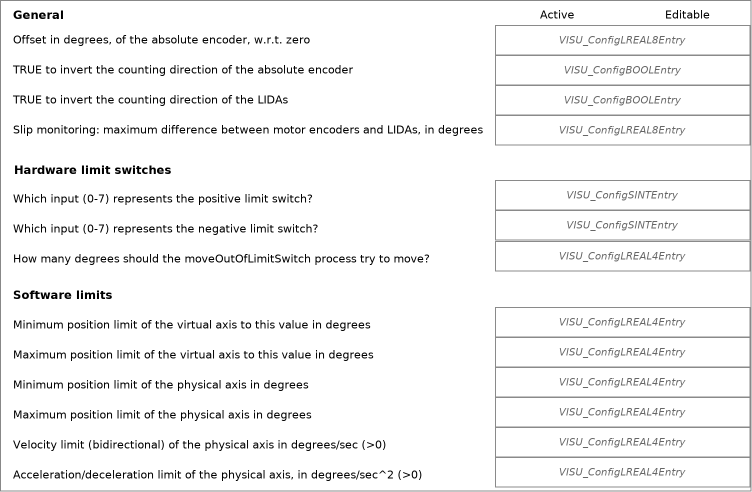
VISUALIZATION VISU_AxesConfig_Elevation_1  // 752x492
VAR_IN_OUT
    active : AxesElevationConfig;
    editable : AxesElevationConfig;
END_VAR
    Label (495,5 125x20), "Active"
    Label (625,5 125x20), "Editable"
    Label (10,25 360x30), "Offset in degrees, of the absolute encoder, w.r.t. zero"
    Frame (495,25 255x30)
        shows VISU_ConfigLREAL8Entry(active := active.absoluteEncoderOffset, editable := editable.absoluteEncoderOffset)
    Label (10,184 475x30), "Which input (0-7) represents the positive limit switch?"
    Label (10,214 475x30), "Which input (0-7) represents the negative limit switch?"
    Label (10,244 475x30), "How many degrees should the moveOutOfLimitSwitch process try to move?"
    Label (11,155 150x30), "Hardware limit switches"
    Label (10,310 475x30), "Minimum position limit of the virtual axis to this value in degrees"
    Label (10,280 165x30), "Software limits"
    Label (10,340 475x30), "Maximum position limit of the virtual axis to this value in degrees"
    Label (10,370 475x30), "Minimum position limit of the physical axis in degrees"
    Label (10,400 475x30), "Maximum position limit of the physical axis in degrees"
    Label (10,430 475x30), "Velocity limit (bidirectional) of the physical axis in degrees/sec (>0)"
    Label (10,460 475x30), "Acceleration/deceleration limit of the physical axis, in degrees/sec^2 (>0)"
    Label (10,115 480x30), "Slip monitoring: maximum difference between motor encoders and LIDAs, in degrees"
    Frame (495,115 255x30)
        shows VISU_ConfigLREAL8Entry(active := active.slipLimit, editable := editable.slipLimit)
    Label (10,0 150x30), "General"
    Frame (495,180 255x30)
        shows VISU_ConfigSINTEntry(active := active.positiveLimitSwitchInput, editable := editable.positiveLimitSwitchInput)
    Frame (495,210 255x30)
        shows VISU_ConfigSINTEntry(active := active.negativeLimitSwitchInput, editable := editable.negativeLimitSwitchInput)
    Frame (495,241 255x30)
        shows VISU_ConfigLREAL4Entry(active := active.moveOutOfLimitSwitchDistance, editable := editable.moveOutOfLimitSwitchDistance)
    Frame (495,307 255x30)
        shows VISU_ConfigLREAL4Entry(active := active.minPositionLimitVirtualAxis, editable := editable.minPositionLimitVirtualAxis)
    Frame (495,337 255x30)
        shows VISU_ConfigLREAL4Entry(active := active.maxPositionLimitVirtualAxis, editable := editable.maxPositionLimitVirtualAxis)
    Frame (495,367 255x30)
        shows VISU_ConfigLREAL4Entry(active := active.minPositionLimitPhysicalAxis, editable := editable.minPositionLimitPhysicalAxis)
    Frame (495,397 255x30)
        shows VISU_ConfigLREAL4Entry(active := active.maxPositionLimitPhysicalAxis, editable := editable.maxPositionLimitPhysicalAxis)
    Frame (495,427 255x30)
        shows VISU_ConfigLREAL4Entry(active := active.velocityLimit, editable := editable.velocityLimit)
    Frame (495,457 255x30)
        shows VISU_ConfigLREAL4Entry(active := active.accelerationLimit, editable := editable.accelerationLimit)
    Frame (495,55 255x30)
        shows VISU_ConfigBOOLEntry(active := active.absoluteEncoderInvert, editable := editable.absoluteEncoderInvert)
    Label (10,55 360x30), "TRUE to invert the counting direction of the absolute encoder"
    Frame (495,85 255x30)
        shows VISU_ConfigBOOLEntry(active := active.lidasInvert, editable := editable.lidasInvert)
    Label (10,85 360x30), "TRUE to invert the counting direction of the LIDAs"
END_VISUALIZATION

(* stored: Version 1.1.0.1, ProductVersion 3.1.4019.2
   Visu VISU_AxesConfig_Elevation_1: Id {0903fd1d-0c8b-4df0-979e-9fb4be80cd03} *)
